TYPE
  ST_SystemStatus_ARP : POINTER TO ARRAY [0..C.uiNumRobotForHMI_C] OF ST_SystemStatus;
END_TYPE

(* stored: Version 1.1.0.1, ProductVersion 3.1.4024.12
   DUT ST_SystemStatus_ARP: Id {00dd4491-93f6-4769-ac71-2dccc5e888ec} *)
